// TIA Portal project "test" (V15.1)
// Vorlageprojekt für das Buch mit Zielsystem S7-1200

(* hardware
DEVICE "S7-1200-Station_1"  S7-1200 Station
   slot 0: "Baugruppenträger_0"  Rack  V1.0
   slot 1: "PLC_1"  CPU 1211C DC/DC/DC  6ES7 211-1AE40-0XB0  V4.1
*)

// ===== PLC "PLC_1"  CPU 1211C DC/DC/DC =====

VAR_GLOBAL   // PLC tag table "Standard-Variablentabelle"
   "Đèn báo hệ thống" AT %A0.0 : Bool;
   "START" AT %E0.0 : Bool;
   "STOP" AT %E0.1 : Bool;
   "Fill_1" AT %QD30 : Real;
   "Cb1" AT %I1.3 : Bool;
   "Lv_1_analog" AT %ID30 : DWord;
   "TG_Run1" AT %M0.0 : Bool;
   "ena_fill_1" AT %M3.0 : Bool;
   "Lv_2_analog" AT %ID34 : DWord;
   "TG_Cb1" AT %M1.3 : Bool;
   "ena_fill_2" AT %M3.4 : Bool;
   "Bt1" AT %Q1.3 : Bool;
   "Fill_2" AT %QD34 : Real;
   "TG_Fill_1" AT %MD30 : Real;
   "TG_Fill_2" AT %MD34 : Real;
   "TG_Fill_3" AT %MD40 : DWord;
   "V3_Calculate_1" AT %MD42 : DWord;
   "Set xa 1" AT %ID38 : Real;
   "Display xa 1" AT %QD54 : DInt;
   "Tag_14" AT %MD54 : DInt;
   "Set xa 2" AT %ID42 : Real;
   "Display xa 2" AT %QD58 : DInt;
   "Level_1" AT %MD10 : Real;
   "TG_Xa1+Xa2" AT %MD0 : DInt;
   "TG_Weight" AT %MD26 : DWord;
   "V3_Calculate" AT %MD38 : Real;
   "V1" AT %MD48 : Real;
   "V2" AT %MD52 : Real;
   "Start_tron" AT %I0.2 : Bool;
   "Tag_1" AT %MW0 : Int;
   "ĐK_Dis_1_2" AT %M1.2 : Bool;
   "Đèn_Trộn_Vàng" AT %Q0.1 : Bool;
   "Red light" AT %Q0.2 : Bool;
   "V3" AT %MD56 : Real;
   "Lv_3_analog" AT %ID46 : Real;
   "Fill_3" AT %QD38 : DWord;
   "TG_Tron_3" AT %M0.2 : Bool;
   "ena_fill_3" AT %M3.6 : Bool;
   "TG_Set1" AT %MD46 : Real;
   "Level_3" AT %MD6 : DInt;
   "Level_2" AT %MD8 : Real;
   "V1_Calculate" AT %MD12 : Real;
   "V2_Calculate" AT %MD16 : Real;
   "Discharge 1" AT %QD42 : Real;
   "Discharge 2" AT %QD46 : Real;
   "ena_discharge_1_2" AT %M3.7 : Bool;
   "TG_Xa_1_2" AT %M0.3 : Bool;
   "Cvey_Weight_1" AT %Q0.5 : Bool;
   "Weight 1" AT %ID50 : Real;
   "m3_Obj_1" AT %MD20 : Real;
   "Discharge 3" AT %QD50 : Real;
   "Start_Chiet" AT %M4.0 : Bool;
   "TG Dis 3" AT %MD50 : Real;
   "Continue with 10kg" AT %M4.1 : Bool;
   "V3_after" AT %MD44 : Real;
   "m3_before" AT %MD58 : DInt;
   "V3_bđầu" AT %MD4 : Real;
   "Tag_3" AT %M5.5 : Bool;
   "Tag_4" AT %M5.6 : Bool;
   "bt2" AT %Q1.4 : Bool;
   "bt3" AT %Q1.5 : Bool;
   "bt4" AT %Q1.6 : Bool;
   "bt5" AT %Q1.7 : Bool;
   "Tag_7" AT %MD28 : DWord;
   "Cb 2" AT %I1.4 : Bool;
   "Tag_9" AT %M10.2 : Bool;
   "Tag_10" AT %MB10 : Byte;
   "Tag_11" AT %M11.0 : Bool;
   "Tag_12" AT %M8.0 : Bool;
   "Tag_15" AT %M20.0 : Bool;
   "Tag_16" AT %M50.0 : Bool;
   "Tag_17" AT %M50.1 : Bool;
   "Wheel On" AT %Q0.6 : Bool;
   "Wheel Left" AT %Q0.7 : Bool;
   "Wheel Right" AT %Q1.0 : Bool;
   "Tag_21" AT %I6.0 : Bool;
   "Tag_22" AT %I6.1 : Bool;
   "Tag_23" AT %M8.5 : Bool;
   "Tag_25" AT %M50.2 : Bool;
   "Tag_26" AT %M50.3 : Bool;
   "Tag_27" AT %M70.1 : Bool;
   "Tag_28" AT %M70.2 : Bool;
   "Cvey_Weight_2" AT %Q0.4 : Bool;
   "Weight 2" AT %ID54 : Real;
   "m3_Obj_2" AT %MD22 : Real;
   "Tag_29" AT %M1.4 : Bool;
   "Tag_30" AT %MW50 : Int;
   "10kg" AT %M40.0 : Bool;
   "15Kg(1)" AT %M40.1 : Bool;
   "Tag_5" AT %M60.0 : Bool;
   "Tag_13" AT %M60.1 : Bool;
   "Tag_18" AT %M60.2 : Bool;
   "Continue with 15kg" AT %M4.2 : Bool;
   "Tag_20" AT %MW30 : Int;
   "STOP when low" AT %M4.3 : Bool;
END_VAR

DATA_BLOCK "ConV Height Volume_DB"   // DB1
{ S7_Optimized_Access := 'TRUE' }
VERSION : 0.1
// stored: InstanceOfName ConV Height Volume
"ConV Height Volume"
BEGIN
END_DATA_BLOCK

DATA_BLOCK "Speed V1 V2_DB"   // DB2
{ S7_Optimized_Access := 'TRUE' }
VERSION : 0.1
// stored: InstanceOfName Speed V1 V2
"Speed V1 V2"
BEGIN
END_DATA_BLOCK

DATA_BLOCK "Dieu kien_DB"   // DB4
{ S7_Optimized_Access := 'TRUE' }
VERSION : 0.1
// stored: InstanceOfName Dieu kien
"Dieu kien"
BEGIN
END_DATA_BLOCK

DATA_BLOCK "Speed V3_DB"   // DB5
{ S7_Optimized_Access := 'TRUE' }
VERSION : 0.1
// stored: InstanceOfName Speed V3
"Speed V3"
BEGIN
END_DATA_BLOCK

// folder: System blocks/Program resources

DATA_BLOCK "T2"   // DB7
{ S7_Optimized_Access := 'TRUE' }
AUTHOR : Simatic
FAMILY : IEC
NAME : IEC_TMR
VERSION : 1.0
// stored: InstanceOfName IEC_TIMER
"IEC_TIMER"
BEGIN
END_DATA_BLOCK

DATA_BLOCK "T3"   // DB8
{ S7_Optimized_Access := 'TRUE' }
AUTHOR : Simatic
FAMILY : IEC
NAME : IEC_TMR
VERSION : 1.0
// stored: InstanceOfName IEC_TIMER
"IEC_TIMER"
BEGIN
END_DATA_BLOCK

// folder: (top level)

FUNCTION_BLOCK "ConV Height Volume"   // FB1, LAD
{ S7_Optimized_Access := 'TRUE' }
VERSION : 0.1
   VAR_INPUT
      AnalogInput1 : Real;
      AnalogInput2 : Real;
      AnalogInput3 : Real;
   END_VAR
   VAR_OUTPUT
      RealLevel1 : Real;
      RealLevel2 : Real;
      RealLevel3 : Real;
      V1 : Real;
      V2 : Real;
      V3 : Real;
   END_VAR
   VAR_TEMP
      AnalogTemp1 : Real;
      AnalogTemp2 : Real;
      AnalogTemp3 : Real;
   END_VAR
BEGIN

REGION Network 1
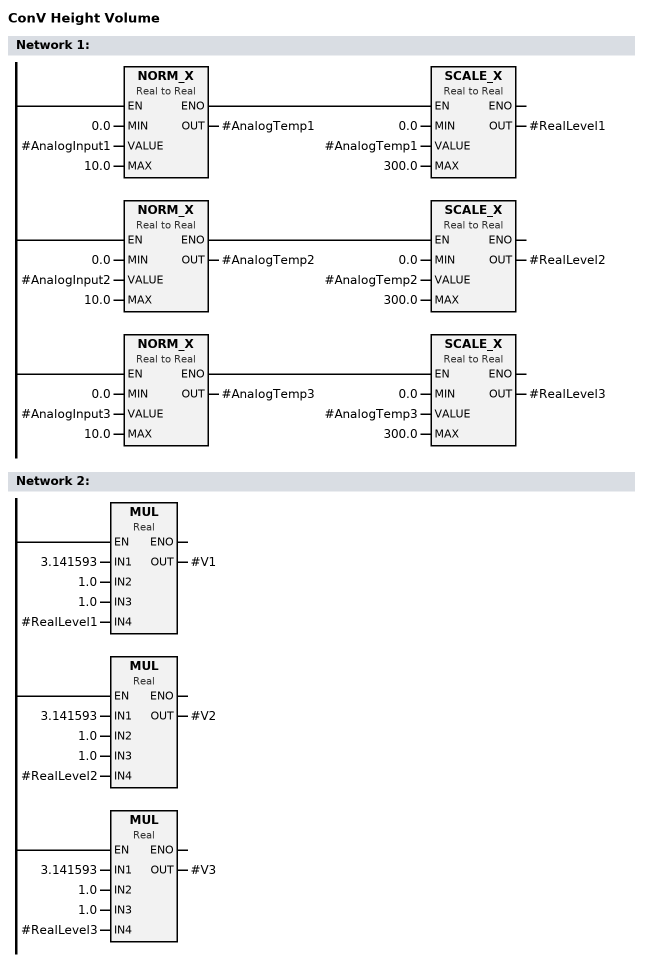
   RUNG wire#powerrail
      { S7_Templates := "[SrcType := Real, DestType := Real]" } Normalize(min := 0.0, value := #AnalogInput1, max := 10.0, out => #AnalogTemp1)
      { S7_Templates := "[SrcType := Real, DestType := Real]" } Scale(min := 0.0, value := #AnalogTemp1, max := 300.0, out => #RealLevel1)
   END_RUNG
   RUNG wire#powerrail
      { S7_Templates := "[SrcType := Real, DestType := Real]" } Normalize(min := 0.0, value := #AnalogInput2, max := 10.0, out => #AnalogTemp2)
      { S7_Templates := "[SrcType := Real, DestType := Real]" } Scale(min := 0.0, value := #AnalogTemp2, max := 300.0, out => #RealLevel2)
   END_RUNG
   RUNG wire#powerrail
      { S7_Templates := "[SrcType := Real, DestType := Real]" } Normalize(min := 0.0, value := #AnalogInput3, max := 10.0, out => #AnalogTemp3)
      { S7_Templates := "[SrcType := Real, DestType := Real]" } Scale(min := 0.0, value := #AnalogTemp3, max := 300.0, out => #RealLevel3)
   END_RUNG
   // the same network as SCL:
   #AnalogTemp1 := NORM_X(MIN := 0.0, VALUE := #AnalogInput1, MAX := 10.0);
   #RealLevel1 := SCALE_X(MIN := 0.0, VALUE := #AnalogTemp1, MAX := 300.0);
   #AnalogTemp2 := NORM_X(MIN := 0.0, VALUE := #AnalogInput2, MAX := 10.0);
   #RealLevel2 := SCALE_X(MIN := 0.0, VALUE := #AnalogTemp2, MAX := 300.0);
   #AnalogTemp3 := NORM_X(MIN := 0.0, VALUE := #AnalogInput3, MAX := 10.0);
   #RealLevel3 := SCALE_X(MIN := 0.0, VALUE := #AnalogTemp3, MAX := 300.0);
END_REGION

REGION Network 2
   RUNG wire#powerrail
      { S7_Templates := "SrcType := Real" } Mul(in1 := 3.141593, in2 := 1.0, in3 := 1.0, in4 := #RealLevel1, out => #V1)
   END_RUNG
   RUNG wire#powerrail
      { S7_Templates := "SrcType := Real" } Mul(in1 := 3.141593, in2 := 1.0, in3 := 1.0, in4 := #RealLevel2, out => #V2)
   END_RUNG
   RUNG wire#powerrail
      { S7_Templates := "SrcType := Real" } Mul(in1 := 3.141593, in2 := 1.0, in3 := 1.0, in4 := #RealLevel3, out => #V3)
   END_RUNG
   // the same network as SCL:
   #V1 := 3.141593 * 1.0 * 1.0 * #RealLevel1;
   #V2 := 3.141593 * 1.0 * 1.0 * #RealLevel2;
   #V3 := 3.141593 * 1.0 * 1.0 * #RealLevel3;
END_REGION
END_FUNCTION_BLOCK

FUNCTION_BLOCK "Dieu kien"   // FB2, LAD
{ S7_Optimized_Access := 'TRUE' }
VERSION : 0.1
   VAR_INPUT
      Display_xa_1 : DInt;
      Display_xa_2 : DInt;
   END_VAR
   VAR_OUTPUT
      V3_calculate : Real;
      V1_Cal : Real;
      V2_Cal : Real;
   END_VAR
   VAR_TEMP
      "int1+int2" : DInt;
      dk1 : Real;   // 100
      dk2 : Real;   // 942.4777 - Thể tích max
      V3_calculate_1 : Real;
      V1_calculate : Real;
      V2_calculate : Real;
   END_VAR
   VAR_TEMP   // added for the SCL form of the ladder/FBD networks
      _w1 : Bool;
      _w2 : Bool;
   END_VAR
BEGIN

REGION Network 1
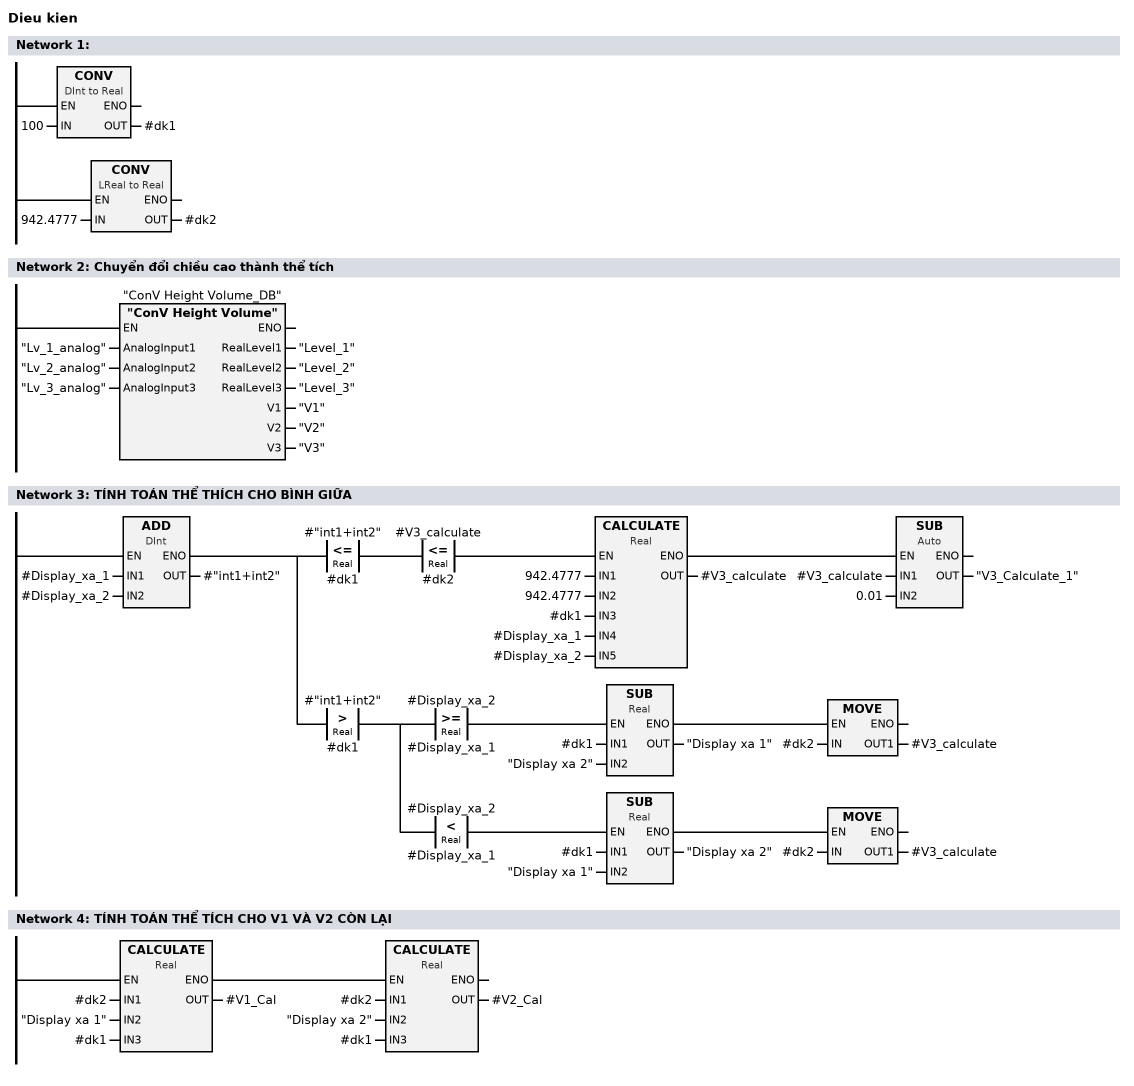
   RUNG wire#powerrail
      { S7_Templates := "[SrcType := DInt, DestType := Real]" } Convert(in := 100, out => #dk1)
   END_RUNG
   RUNG wire#powerrail
      { S7_Templates := "[SrcType := LReal, DestType := Real]" } Convert(in := 942.4777, out => #dk2)
   END_RUNG
   // the same network as SCL:
   #dk1 := DINT_TO_REAL(100);
   #dk2 := LREAL_TO_REAL(942.4777);
END_REGION

REGION Network 2: Chuyển đổi chiều cao thành thể tích
   RUNG wire#powerrail
      "ConV Height Volume_DB"(AnalogInput1 := "Lv_1_analog", AnalogInput2 := "Lv_2_analog", AnalogInput3 := "Lv_3_analog", RealLevel1 => "Level_1", RealLevel2 => "Level_2", RealLevel3 => "Level_3", V1 => "V1", V2 => "V2", V3 => "V3")
   END_RUNG
   // the same network as SCL:
   "ConV Height Volume_DB"(AnalogInput1 := "Lv_1_analog",   // "ConV Height Volume"
                           AnalogInput2 := "Lv_2_analog",
                           AnalogInput3 := "Lv_3_analog",
                           RealLevel1 => "Level_1",
                           RealLevel2 => "Level_2",
                           RealLevel3 => "Level_3",
                           V1 => "V1",
                           V2 => "V2",
                           V3 => "V3");
END_REGION

REGION Network 3: TÍNH TOÁN THỂ THÍCH CHO BÌNH GIỮA
   RUNG wire#powerrail
      { S7_Templates := "SrcType := DInt" } Add(in1 := #Display_xa_1, in2 := #Display_xa_2, out => #"int1+int2")
      wire#w1
      { S7_Templates := "SrcType := Real" } LE_Contact(in1 := #"int1+int2", in2 := #dk1)
      { S7_Templates := "SrcType := Real" } LE_Contact(in1 := #V3_calculate, in2 := #dk2)
      { S7_Templates := "SrcType := Real"; S7_Expression := "IN1*IN4/IN3+IN2*IN5/IN3" } Calculate(in1 := 942.4777, in2 := 942.4777, in3 := #dk1, in4 := #Display_xa_1, in5 := #Display_xa_2, out => #V3_calculate)
      Sub(in1 := #V3_calculate, in2 := 0.01, out => "V3_Calculate_1")
   END_RUNG
   RUNG wire#w1
      { S7_Templates := "SrcType := Real" } GT_Contact(in1 := #"int1+int2", in2 := #dk1)
      wire#w2
      { S7_Templates := "SrcType := Real" } GE_Contact(in1 := #Display_xa_2, in2 := #Display_xa_1)
      { S7_Templates := "SrcType := Real" } Sub(in1 := #dk1, in2 := "Display xa 2", out => "Display xa 1")
      Move(in := #dk2, out1 => #V3_calculate)
   END_RUNG
   RUNG wire#w2
      { S7_Templates := "SrcType := Real" } LT_Contact(in1 := #Display_xa_2, in2 := #Display_xa_1)
      { S7_Templates := "SrcType := Real" } Sub(in1 := #dk1, in2 := "Display xa 1", out => "Display xa 2")
      Move(in := #dk2, out1 => #V3_calculate)
   END_RUNG
   // the same network as SCL:
   #"int1+int2" := #Display_xa_1 + #Display_xa_2;
   #_w1 := (#"int1+int2" <= #dk1) AND (#V3_calculate <= #dk2);
   IF #_w1 THEN
       #V3_calculate := 942.4777*#Display_xa_1/#dk1+942.4777*#Display_xa_2/#dk1;
       "V3_Calculate_1" := #V3_calculate - 0.01;
   END_IF;
   #_w2 := #"int1+int2" > #dk1;
   IF #_w2 AND (#Display_xa_2 >= #Display_xa_1) THEN
       "Display xa 1" := #dk1 - "Display xa 2";
       #V3_calculate := #dk2;
   END_IF;
   IF #_w2 AND (#Display_xa_2 < #Display_xa_1) THEN
       "Display xa 2" := #dk1 - "Display xa 1";
       #V3_calculate := #dk2;
   END_IF;
END_REGION

REGION Network 4: TÍNH TOÁN THỂ TÍCH CHO V1 VÀ V2 CÒN LẠI
   RUNG wire#powerrail
      { S7_Templates := "SrcType := Real"; S7_Expression := "(IN1-IN2*IN1/IN3)" } Calculate(in1 := #dk2, in2 := "Display xa 1", in3 := #dk1, out => #V1_Cal)
      { S7_Templates := "SrcType := Real"; S7_Expression := "(IN1-IN2*IN1/IN3)" } Calculate(in1 := #dk2, in2 := "Display xa 2", in3 := #dk1, out => #V2_Cal)
   END_RUNG
   // the same network as SCL:
   #V1_Cal := (#dk2-"Display xa 1"*#dk2/#dk1);
   #V2_Cal := (#dk2-"Display xa 2"*#dk2/#dk1);
END_REGION
END_FUNCTION_BLOCK

FUNCTION_BLOCK "Speed V3"   // FB3, LAD
{ S7_Optimized_Access := 'TRUE' }
VERSION : 0.1
   VAR_OUTPUT
      "Speed Fill 3" : Real;
   END_VAR
   VAR_TEMP
      dk1 : DInt;   // 150
      hs1 : DInt;   // 490
      dk2 : DInt;   // 295
      hs2 : DInt;   // 10
      Temp_1 : DInt;
      "Speed Fill 3 Dint" : Real;
      V3_Calculate : Real;
   END_VAR
BEGIN

REGION Network 1
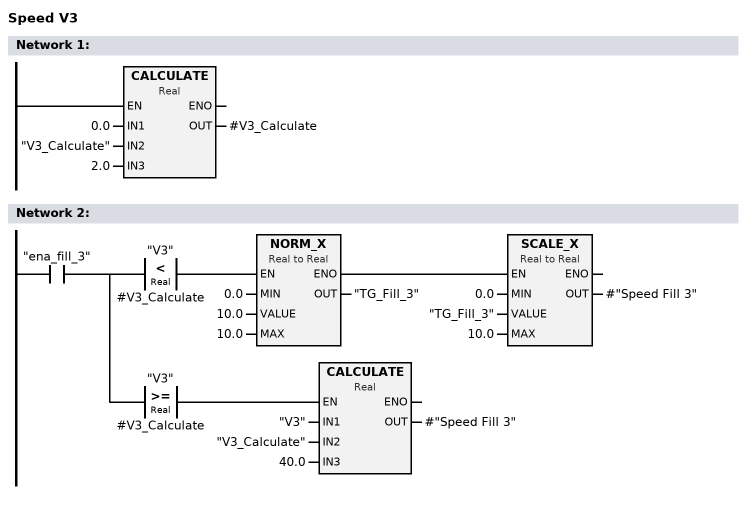
   RUNG wire#powerrail
      { S7_Templates := "SrcType := Real"; S7_Expression := "(IN2-IN1)/IN3" } Calculate(in1 := 0.0, in2 := "V3_Calculate", in3 := 2.0, out => #V3_Calculate)
   END_RUNG
   // the same network as SCL:
   #V3_Calculate := ("V3_Calculate"-0.0)/2.0;
END_REGION

REGION Network 2
   RUNG wire#powerrail
      Contact( "ena_fill_3" )
      wire#w1
      { S7_Templates := "SrcType := Real" } LT_Contact(in1 := "V3", in2 := #V3_Calculate)
      { S7_Templates := "[SrcType := Real, DestType := Real]" } Normalize(min := 0.0, value := 10.0, max := 10.0, out => "TG_Fill_3")
      { S7_Templates := "[SrcType := Real, DestType := Real]" } Scale(min := 0.0, value := "TG_Fill_3", max := 10.0, out => #"Speed Fill 3")
   END_RUNG
   RUNG wire#w1
      { S7_Templates := "SrcType := Real" } GE_Contact(in1 := "V3", in2 := #V3_Calculate)
      { S7_Templates := "SrcType := Real"; S7_Expression := "-IN3*IN1*IN1/(IN2*IN2)+IN3*IN1/IN2" } Calculate(in1 := "V3", in2 := "V3_Calculate", in3 := 40.0, out => #"Speed Fill 3")
   END_RUNG
   // the same network as SCL:
   IF "ena_fill_3" AND ("V3" < #V3_Calculate) THEN
       "TG_Fill_3" := NORM_X(MIN := 0.0, VALUE := 10.0, MAX := 10.0);
       #"Speed Fill 3" := SCALE_X(MIN := 0.0, VALUE := "TG_Fill_3", MAX := 10.0);
   END_IF;
   IF "ena_fill_3" AND ("V3" >= #V3_Calculate) THEN
       #"Speed Fill 3" := -40.0*"V3"*"V3"/("V3_Calculate"*"V3_Calculate")+40.0*"V3"/"V3_Calculate";
   END_IF;
END_REGION
END_FUNCTION_BLOCK

FUNCTION_BLOCK "Speed V1 V2"   // FB4, LAD
{ S7_Optimized_Access := 'TRUE' }
VERSION : 0.1
   VAR_OUTPUT
      "Speed dis 1" : Real;
      "Speed dis 2" : Real;
   END_VAR
   VAR_TEMP
      V1_Calculate : Real;
      V2_Calculate : Real;
      TG_Dis_1 : DWord;
      TG_Dis_2 : DWord;
   END_VAR
BEGIN

REGION Network 1
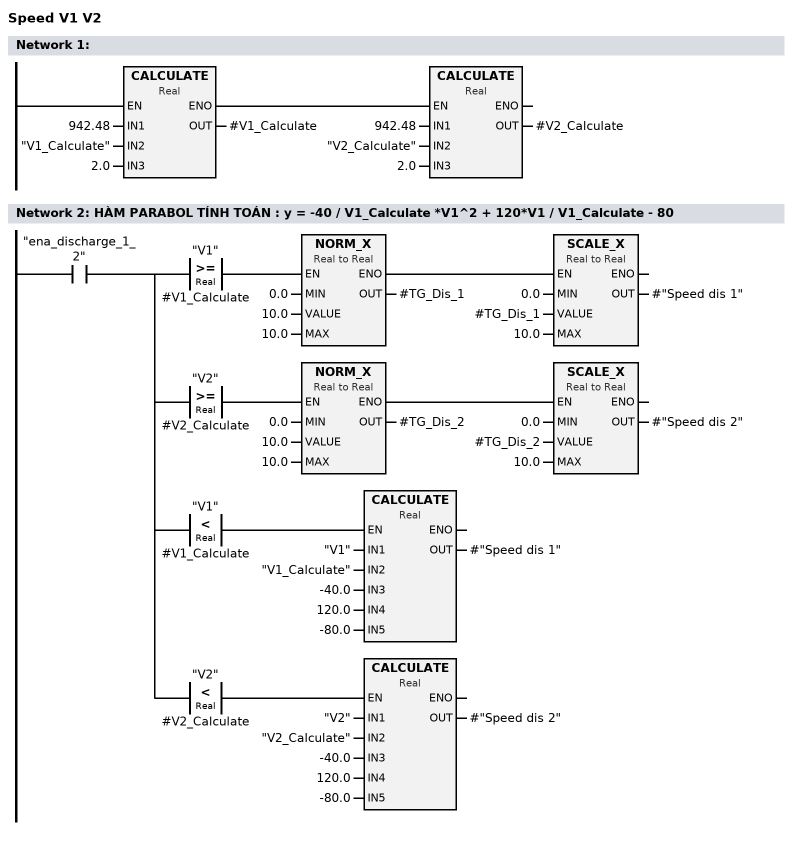
   RUNG wire#powerrail
      { S7_Templates := "SrcType := Real"; S7_Expression := "(IN1-IN2)/IN3+IN2" } Calculate(in1 := 942.48, in2 := "V1_Calculate", in3 := 2.0, out => #V1_Calculate)
      { S7_Templates := "SrcType := Real"; S7_Expression := "(IN1-IN2)/IN3+IN2" } Calculate(in1 := 942.48, in2 := "V2_Calculate", in3 := 2.0, out => #V2_Calculate)
   END_RUNG
   // the same network as SCL:
   #V1_Calculate := (942.48-"V1_Calculate")/2.0+"V1_Calculate";
   #V2_Calculate := (942.48-"V2_Calculate")/2.0+"V2_Calculate";
END_REGION

REGION Network 2: HÀM PARABOL TÍNH TOÁN : y = -40 / V1_Calculate *V1^2 + 120*V1 / V1_Calculate - 80
   RUNG wire#powerrail
      Contact( "ena_discharge_1_2" )
      wire#w1
      { S7_Templates := "SrcType := Real" } GE_Contact(in1 := "V1", in2 := #V1_Calculate)
      { S7_Templates := "[SrcType := Real, DestType := Real]" } Normalize(min := 0.0, value := 10.0, max := 10.0, out => #TG_Dis_1)
      { S7_Templates := "[SrcType := Real, DestType := Real]" } Scale(min := 0.0, value := #TG_Dis_1, max := 10.0, out => #"Speed dis 1")
   END_RUNG
   RUNG wire#w1
      { S7_Templates := "SrcType := Real" } GE_Contact(in1 := "V2", in2 := #V2_Calculate)
      { S7_Templates := "[SrcType := Real, DestType := Real]" } Normalize(min := 0.0, value := 10.0, max := 10.0, out => #TG_Dis_2)
      { S7_Templates := "[SrcType := Real, DestType := Real]" } Scale(min := 0.0, value := #TG_Dis_2, max := 10.0, out => #"Speed dis 2")
   END_RUNG
   RUNG wire#w1
      { S7_Templates := "SrcType := Real" } LT_Contact(in1 := "V1", in2 := #V1_Calculate)
      { S7_Templates := "SrcType := Real"; S7_Expression := "IN3/(IN2*IN2)*IN1*IN1+IN4*IN1/IN2+IN5" } Calculate(in1 := "V1", in2 := "V1_Calculate", in3 := -40.0, in4 := 120.0, in5 := -80.0, out => #"Speed dis 1")
   END_RUNG
   RUNG wire#w1
      { S7_Templates := "SrcType := Real" } LT_Contact(in1 := "V2", in2 := #V2_Calculate)
      { S7_Templates := "SrcType := Real"; S7_Expression := "IN3/(IN2*IN2)*IN1*IN1+IN4*IN1/IN2+IN5" } Calculate(in1 := "V2", in2 := "V2_Calculate", in3 := -40.0, in4 := 120.0, in5 := -80.0, out => #"Speed dis 2")
   END_RUNG
   // the same network as SCL:
   IF "ena_discharge_1_2" AND ("V1" >= #V1_Calculate) THEN
       #TG_Dis_1 := NORM_X(MIN := 0.0, VALUE := 10.0, MAX := 10.0);
       #"Speed dis 1" := SCALE_X(MIN := 0.0, VALUE := #TG_Dis_1, MAX := 10.0);
   END_IF;
   IF "ena_discharge_1_2" AND ("V2" >= #V2_Calculate) THEN
       #TG_Dis_2 := NORM_X(MIN := 0.0, VALUE := 10.0, MAX := 10.0);
       #"Speed dis 2" := SCALE_X(MIN := 0.0, VALUE := #TG_Dis_2, MAX := 10.0);
   END_IF;
   IF "ena_discharge_1_2" AND ("V1" < #V1_Calculate) THEN
       #"Speed dis 1" := (-40.0)/("V1_Calculate"*"V1_Calculate")*"V1"*"V1"+120.0*"V1"/"V1_Calculate"+(-80.0);
   END_IF;
   IF "ena_discharge_1_2" AND ("V2" < #V2_Calculate) THEN
       #"Speed dis 2" := (-40.0)/("V2_Calculate"*"V2_Calculate")*"V2"*"V2"+120.0*"V2"/"V2_Calculate"+(-80.0);
   END_IF;
END_REGION
END_FUNCTION_BLOCK

FUNCTION "Run" : Void   // FC1, LAD
{ S7_Optimized_Access := 'TRUE' }
VERSION : 0.1
BEGIN

REGION Network 1
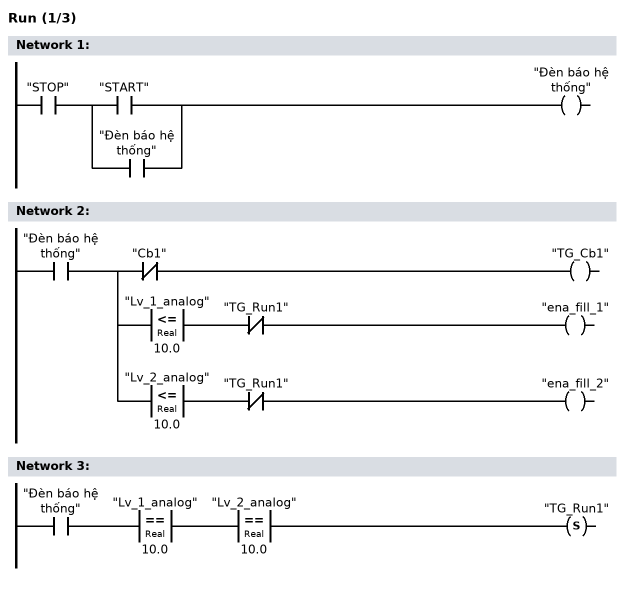
   RUNG wire#powerrail
      Contact( "STOP" )
      wire#w1
      Contact( "START" )
      wire#w2
      Coil( "Đèn báo hệ thống" )
   END_RUNG
   RUNG wire#w1
      Contact( "Đèn báo hệ thống" )
   END_RUNG wire#w2
   // the same network as SCL:
   "Đèn báo hệ thống" := "STOP" AND ("START" OR "Đèn báo hệ thống");
END_REGION

REGION Network 2
   RUNG wire#powerrail
      Contact( "Đèn báo hệ thống" )
      wire#w1
      I_Contact( "Cb1" )
      Coil( "TG_Cb1" )
   END_RUNG
   RUNG wire#w1
      { S7_Templates := "SrcType := Real" } LE_Contact(in1 := "Lv_1_analog", in2 := 10.0)
      I_Contact( "TG_Run1" )
      Coil( "ena_fill_1" )
   END_RUNG
   RUNG wire#w1
      { S7_Templates := "SrcType := Real" } LE_Contact(in1 := "Lv_2_analog", in2 := 10.0)
      I_Contact( "TG_Run1" )
      Coil( "ena_fill_2" )
   END_RUNG
   // the same network as SCL:
   "TG_Cb1" := "Đèn báo hệ thống" AND NOT "Cb1";
   "ena_fill_1" := "Đèn báo hệ thống" AND ("Lv_1_analog" <= 10.0) AND NOT "TG_Run1";
   "ena_fill_2" := "Đèn báo hệ thống" AND ("Lv_2_analog" <= 10.0) AND NOT "TG_Run1";
END_REGION

REGION Network 3
   RUNG wire#powerrail
      Contact( "Đèn báo hệ thống" )
      { S7_Templates := "SrcType := Real" } EQ_Contact(in1 := "Lv_1_analog", in2 := 10.0)
      { S7_Templates := "SrcType := Real" } EQ_Contact(in1 := "Lv_2_analog", in2 := 10.0)
      S_Coil( "TG_Run1" )
   END_RUNG
   // the same network as SCL:
   IF "Đèn báo hệ thống" AND ("Lv_1_analog" = 10.0) AND ("Lv_2_analog" = 10.0) THEN
       "TG_Run1" := TRUE;
   END_IF;
END_REGION

REGION Network 4
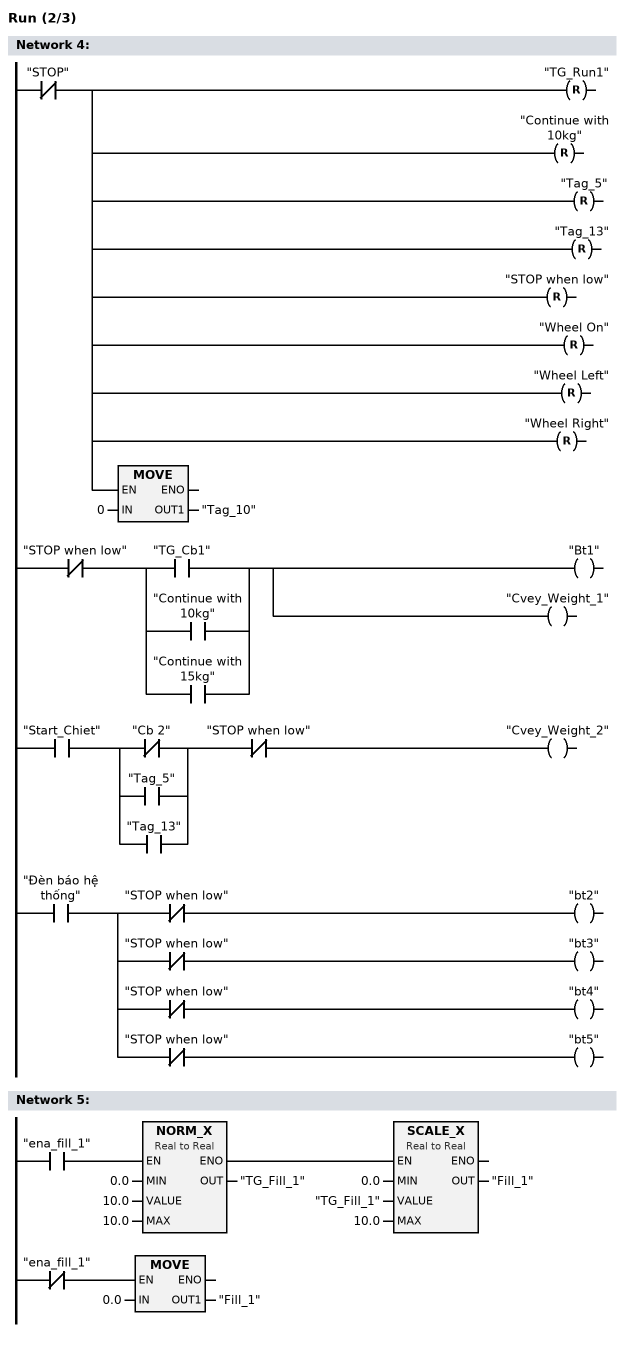
   RUNG wire#powerrail
      I_Contact( "STOP" )
      wire#w1
      R_Coil( "TG_Run1" )
   END_RUNG
   RUNG wire#w1
      R_Coil( "Continue with 10kg" )
   END_RUNG
   RUNG wire#w1
      R_Coil( "Tag_5" )
   END_RUNG
   RUNG wire#w1
      R_Coil( "Tag_13" )
   END_RUNG
   RUNG wire#w1
      R_Coil( "STOP when low" )
   END_RUNG
   RUNG wire#w1
      R_Coil( "Wheel On" )
   END_RUNG
   RUNG wire#w1
      R_Coil( "Wheel Left" )
   END_RUNG
   RUNG wire#w1
      R_Coil( "Wheel Right" )
   END_RUNG
   RUNG wire#w1
      Move(in := 0, out1 => "Tag_10")
   END_RUNG
   RUNG wire#powerrail
      I_Contact( "STOP when low" )
      wire#w2
      Contact( "TG_Cb1" )
      wire#w3
      Coil( "Bt1" )
   END_RUNG
   RUNG wire#w2
      Contact( "Continue with 10kg" )
   END_RUNG wire#w3
   RUNG wire#w2
      Contact( "Continue with 15kg" )
   END_RUNG wire#w3
   RUNG wire#w3
      Coil( "Cvey_Weight_1" )
   END_RUNG
   RUNG wire#powerrail
      Contact( "Start_Chiet" )
      wire#w4
      I_Contact( "Cb 2" )
      wire#w5
      I_Contact( "STOP when low" )
      Coil( "Cvey_Weight_2" )
   END_RUNG
   RUNG wire#w4
      Contact( "Tag_5" )
   END_RUNG wire#w5
   RUNG wire#w4
      Contact( "Tag_13" )
   END_RUNG wire#w5
   RUNG wire#powerrail
      Contact( "Đèn báo hệ thống" )
      wire#w6
      I_Contact( "STOP when low" )
      Coil( "bt2" )
   END_RUNG
   RUNG wire#w6
      I_Contact( "STOP when low" )
      Coil( "bt3" )
   END_RUNG
   RUNG wire#w6
      I_Contact( "STOP when low" )
      Coil( "bt4" )
   END_RUNG
   RUNG wire#w6
      I_Contact( "STOP when low" )
      Coil( "bt5" )
   END_RUNG
   // the same network as SCL:
   IF NOT "STOP" THEN
       "TG_Run1" := FALSE;
       "Continue with 10kg" := FALSE;
       "Tag_5" := FALSE;
       "Tag_13" := FALSE;
       "STOP when low" := FALSE;
       "Wheel On" := FALSE;
       "Wheel Left" := FALSE;
       "Wheel Right" := FALSE;
       "Tag_10" := 0;
   END_IF;
   "Bt1" := NOT "STOP when low" AND ("TG_Cb1" OR "Continue with 10kg" OR "Continue with 15kg");
   "Cvey_Weight_1" := "Bt1";
   "Cvey_Weight_2" := "Start_Chiet" AND (NOT "Cb 2" OR "Tag_5" OR "Tag_13") AND NOT "STOP when low";
   "bt2" := "Đèn báo hệ thống" AND NOT "STOP when low";
   "bt3" := "Đèn báo hệ thống" AND NOT "STOP when low";
   "bt4" := "Đèn báo hệ thống" AND NOT "STOP when low";
   "bt5" := "Đèn báo hệ thống" AND NOT "STOP when low";
END_REGION

REGION Network 5
   RUNG wire#powerrail
      Contact( "ena_fill_1" )
      { S7_Templates := "[SrcType := Real, DestType := Real]" } Normalize(min := 0.0, value := 10.0, max := 10.0, out => "TG_Fill_1")
      { S7_Templates := "[SrcType := Real, DestType := Real]" } Scale(min := 0.0, value := "TG_Fill_1", max := 10.0, out => "Fill_1")
   END_RUNG
   RUNG wire#powerrail
      I_Contact( "ena_fill_1" )
      Move(in := 0.0, out1 => "Fill_1")
   END_RUNG
   // the same network as SCL:
   IF "ena_fill_1" THEN
       "TG_Fill_1" := NORM_X(MIN := 0.0, VALUE := 10.0, MAX := 10.0);
       "Fill_1" := SCALE_X(MIN := 0.0, VALUE := "TG_Fill_1", MAX := 10.0);
   END_IF;
   IF NOT "ena_fill_1" THEN "Fill_1" := 0.0; END_IF;
END_REGION

REGION Network 6
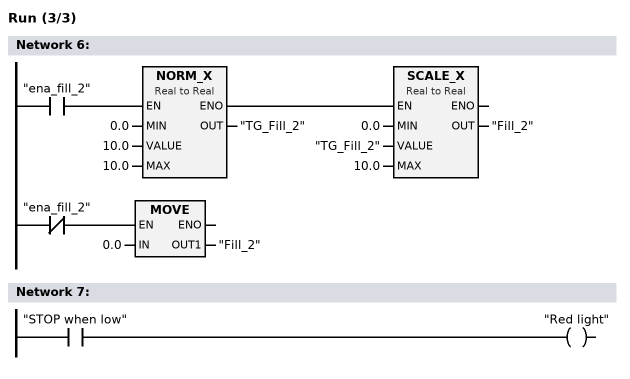
   RUNG wire#powerrail
      Contact( "ena_fill_2" )
      { S7_Templates := "[SrcType := Real, DestType := Real]" } Normalize(min := 0.0, value := 10.0, max := 10.0, out => "TG_Fill_2")
      { S7_Templates := "[SrcType := Real, DestType := Real]" } Scale(min := 0.0, value := "TG_Fill_2", max := 10.0, out => "Fill_2")
   END_RUNG
   RUNG wire#powerrail
      I_Contact( "ena_fill_2" )
      Move(in := 0.0, out1 => "Fill_2")
   END_RUNG
   // the same network as SCL:
   IF "ena_fill_2" THEN
       "TG_Fill_2" := NORM_X(MIN := 0.0, VALUE := 10.0, MAX := 10.0);
       "Fill_2" := SCALE_X(MIN := 0.0, VALUE := "TG_Fill_2", MAX := 10.0);
   END_IF;
   IF NOT "ena_fill_2" THEN "Fill_2" := 0.0; END_IF;
END_REGION

REGION Network 7
   RUNG wire#powerrail
      Contact( "STOP when low" )
      Coil( "Red light" )
   END_RUNG
   // the same network as SCL:
   "Red light" := "STOP when low";
END_REGION
END_FUNCTION

FUNCTION "Tron" : Void   // FC2, LAD
{ S7_Optimized_Access := 'TRUE' }
VERSION : 0.1
   VAR_TEMP   // added for the SCL form of the ladder/FBD networks
      _w1 : Bool;
   END_VAR
BEGIN

REGION Network 1
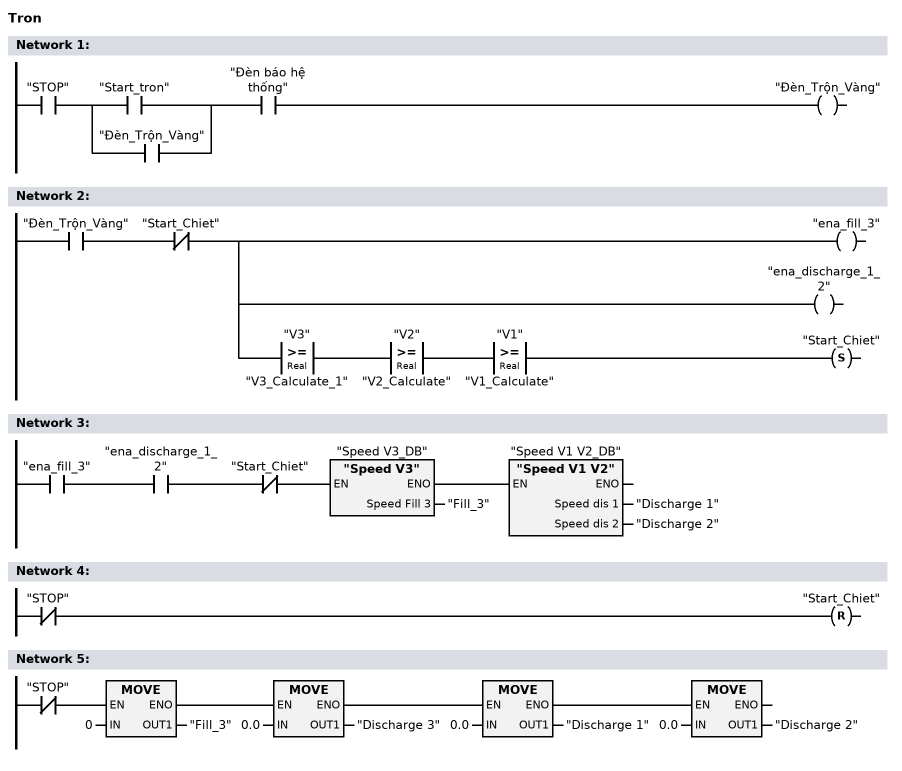
   RUNG wire#powerrail
      Contact( "STOP" )
      wire#w1
      Contact( "Start_tron" )
      wire#w2
      Contact( "Đèn báo hệ thống" )
      Coil( "Đèn_Trộn_Vàng" )
   END_RUNG
   RUNG wire#w1
      Contact( "Đèn_Trộn_Vàng" )
   END_RUNG wire#w2
   // the same network as SCL:
   "Đèn_Trộn_Vàng" := "STOP" AND ("Start_tron" OR "Đèn_Trộn_Vàng") AND "Đèn báo hệ thống";
END_REGION

REGION Network 2
   RUNG wire#powerrail
      Contact( "Đèn_Trộn_Vàng" )
      I_Contact( "Start_Chiet" )
      wire#w1
      Coil( "ena_fill_3" )
   END_RUNG
   RUNG wire#w1
      Coil( "ena_discharge_1_2" )
   END_RUNG
   RUNG wire#w1
      { S7_Templates := "SrcType := Real" } GE_Contact(in1 := "V3", in2 := "V3_Calculate_1")
      { S7_Templates := "SrcType := Real" } GE_Contact(in1 := "V2", in2 := "V2_Calculate")
      { S7_Templates := "SrcType := Real" } GE_Contact(in1 := "V1", in2 := "V1_Calculate")
      S_Coil( "Start_Chiet" )
   END_RUNG
   // the same network as SCL:
   "ena_fill_3" := "Đèn_Trộn_Vàng" AND NOT "Start_Chiet";
   "ena_discharge_1_2" := "ena_fill_3";
   IF "ena_fill_3" AND ("V3" >= "V3_Calculate_1") AND ("V2" >= "V2_Calculate") AND ("V1" >= "V1_Calculate") THEN
       "Start_Chiet" := TRUE;
   END_IF;
END_REGION

REGION Network 3
   RUNG wire#powerrail
      Contact( "ena_fill_3" )
      Contact( "ena_discharge_1_2" )
      I_Contact( "Start_Chiet" )
      "Speed V3_DB"("Speed Fill 3" => "Fill_3")
      "Speed V1 V2_DB"("Speed dis 1" => "Discharge 1", "Speed dis 2" => "Discharge 2")
   END_RUNG
   // the same network as SCL:
   "Speed V3_DB"(EN := "ena_fill_3" AND "ena_discharge_1_2" AND NOT "Start_Chiet",   // "Speed V3"
                 "Speed Fill 3" => "Fill_3",
                 ENO => #_w1);
   IF #_w1 THEN
       "Speed V1 V2_DB"("Speed dis 1" => "Discharge 1", "Speed dis 2" => "Discharge 2");   // "Speed V1 V2"
   END_IF;
END_REGION

REGION Network 4
   RUNG wire#powerrail
      I_Contact( "STOP" )
      R_Coil( "Start_Chiet" )
   END_RUNG
   // the same network as SCL:
   IF NOT "STOP" THEN "Start_Chiet" := FALSE; END_IF;
END_REGION

REGION Network 5
   RUNG wire#powerrail
      I_Contact( "STOP" )
      Move(in := 0, out1 => "Fill_3")
      Move(in := 0.0, out1 => "Discharge 3")
      Move(in := 0.0, out1 => "Discharge 1")
      Move(in := 0.0, out1 => "Discharge 2")
   END_RUNG
   // the same network as SCL:
   IF NOT "STOP" THEN
       "Fill_3" := 0;
       "Discharge 3" := 0.0;
       "Discharge 1" := 0.0;
       "Discharge 2" := 0.0;
   END_IF;
END_REGION
END_FUNCTION

FUNCTION "Hien thi muc Xa" : Void   // FC3, LAD
{ S7_Optimized_Access := 'TRUE' }
VERSION : 0.1
BEGIN

REGION Network 1
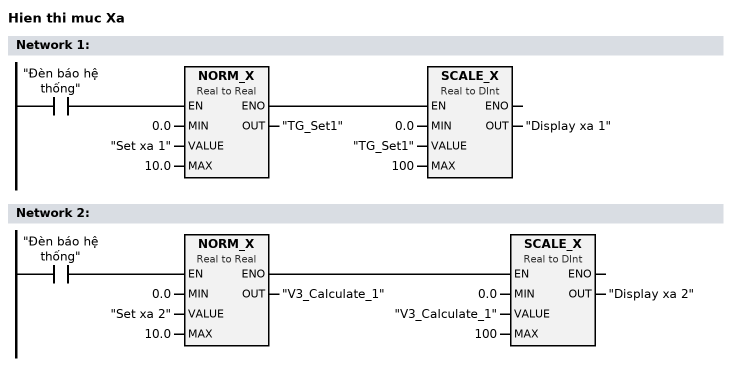
   RUNG wire#powerrail
      Contact( "Đèn báo hệ thống" )
      { S7_Templates := "[SrcType := Real, DestType := Real]" } Normalize(min := 0.0, value := "Set xa 1", max := 10.0, out => "TG_Set1")
      { S7_Templates := "[SrcType := Real, DestType := DInt]" } Scale(min := 0.0, value := "TG_Set1", max := 100, out => "Display xa 1")
   END_RUNG
   // the same network as SCL:
   IF "Đèn báo hệ thống" THEN
       "TG_Set1" := NORM_X(MIN := 0.0, VALUE := "Set xa 1", MAX := 10.0);
       "Display xa 1" := SCALE_X(MIN := 0.0, VALUE := "TG_Set1", MAX := 100);
   END_IF;
END_REGION

REGION Network 2
   RUNG wire#powerrail
      Contact( "Đèn báo hệ thống" )
      { S7_Templates := "[SrcType := Real, DestType := Real]" } Normalize(min := 0.0, value := "Set xa 2", max := 10.0, out => "V3_Calculate_1")
      { S7_Templates := "[SrcType := Real, DestType := DInt]" } Scale(min := 0.0, value := "V3_Calculate_1", max := 100, out => "Display xa 2")
   END_RUNG
   // the same network as SCL:
   IF "Đèn báo hệ thống" THEN
       "V3_Calculate_1" := NORM_X(MIN := 0.0, VALUE := "Set xa 2", MAX := 10.0);
       "Display xa 2" := SCALE_X(MIN := 0.0, VALUE := "V3_Calculate_1", MAX := 100);
   END_IF;
END_REGION
END_FUNCTION

FUNCTION "Sorting and fill" : Void   // FC4, LAD
{ S7_Optimized_Access := 'TRUE' }
VERSION : 0.1
   VAR_TEMP
      Obj_Weight_1 : Real;
      v3_After : Real;
      TG_Dis_3 : Real;
      Obj_Weight_2 : Real;
   END_VAR
   VAR_TEMP   // added for the SCL form of the ladder/FBD networks
      _w1 : Bool;
      _w2 : Bool;
      _w3 : Bool;
   END_VAR
BEGIN

REGION Network 1
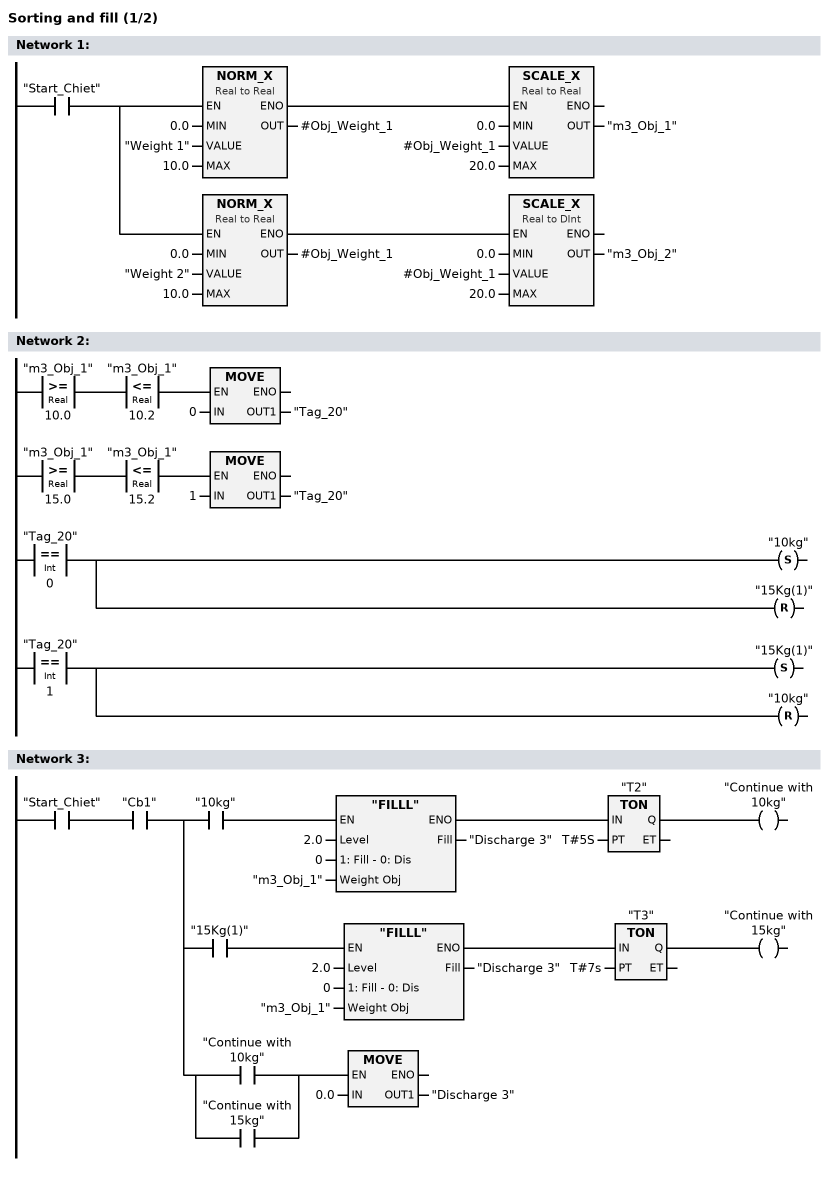
   RUNG wire#powerrail
      Contact( "Start_Chiet" )
      wire#w1
      { S7_Templates := "[SrcType := Real, DestType := Real]" } Normalize(min := 0.0, value := "Weight 1", max := 10.0, out => #Obj_Weight_1)
      { S7_Templates := "[SrcType := Real, DestType := Real]" } Scale(min := 0.0, value := #Obj_Weight_1, max := 20.0, out => "m3_Obj_1")
   END_RUNG
   RUNG wire#w1
      { S7_Templates := "[SrcType := Real, DestType := Real]" } Normalize(min := 0.0, value := "Weight 2", max := 10.0, out => #Obj_Weight_1)
      { S7_Templates := "[SrcType := Real, DestType := DInt]" } Scale(min := 0.0, value := #Obj_Weight_1, max := 20.0, out => "m3_Obj_2")
   END_RUNG
   // the same network as SCL:
   IF "Start_Chiet" THEN
       #Obj_Weight_1 := NORM_X(MIN := 0.0, VALUE := "Weight 1", MAX := 10.0);
       "m3_Obj_1" := SCALE_X(MIN := 0.0, VALUE := #Obj_Weight_1, MAX := 20.0);
       #Obj_Weight_1 := NORM_X(MIN := 0.0, VALUE := "Weight 2", MAX := 10.0);
       "m3_Obj_2" := SCALE_X(MIN := 0.0, VALUE := #Obj_Weight_1, MAX := 20.0);
   END_IF;
END_REGION

REGION Network 2
   RUNG wire#powerrail
      { S7_Templates := "SrcType := Real" } GE_Contact(in1 := "m3_Obj_1", in2 := 10.0)
      { S7_Templates := "SrcType := Real" } LE_Contact(in1 := "m3_Obj_1", in2 := 10.2)
      Move(in := 0, out1 => "Tag_20")
   END_RUNG
   RUNG wire#powerrail
      { S7_Templates := "SrcType := Real" } GE_Contact(in1 := "m3_Obj_1", in2 := 15.0)
      { S7_Templates := "SrcType := Real" } LE_Contact(in1 := "m3_Obj_1", in2 := 15.2)
      Move(in := 1, out1 => "Tag_20")
   END_RUNG
   RUNG wire#powerrail
      { S7_Templates := "SrcType := Int" } EQ_Contact(in1 := "Tag_20", in2 := 0)
      wire#w1
      S_Coil( "10kg" )
   END_RUNG
   RUNG wire#w1
      R_Coil( "15Kg(1)" )
   END_RUNG
   RUNG wire#powerrail
      { S7_Templates := "SrcType := Int" } EQ_Contact(in1 := "Tag_20", in2 := 1)
      wire#w2
      S_Coil( "15Kg(1)" )
   END_RUNG
   RUNG wire#w2
      R_Coil( "10kg" )
   END_RUNG
   // the same network as SCL:
   IF ("m3_Obj_1" >= 10.0) AND ("m3_Obj_1" <= 10.2) THEN "Tag_20" := 0; END_IF;
   IF ("m3_Obj_1" >= 15.0) AND ("m3_Obj_1" <= 15.2) THEN "Tag_20" := 1; END_IF;
   IF "Tag_20" = 0 THEN
       "10kg" := TRUE;
       "15Kg(1)" := FALSE;
   END_IF;
   IF "Tag_20" = 1 THEN
       "15Kg(1)" := TRUE;
       "10kg" := FALSE;
   END_IF;
END_REGION

REGION Network 3
   #_w1 := "Start_Chiet" AND "Cb1";
   "FILLL"(EN := #_w1 AND "10kg",
           Level := 2.0,
           "1: Fill - 0: Dis" := 0,
           "Weight Obj" := "m3_Obj_1",
           Fill => "Discharge 3",
           ENO => #_w2);
   "T2".TON(IN := #_w2, PT := T#5S);
   "Continue with 10kg" := "T2".Q;
   "FILLL"(EN := #_w1 AND "15Kg(1)",
           Level := 2.0,
           "1: Fill - 0: Dis" := 0,
           "Weight Obj" := "m3_Obj_1",
           Fill => "Discharge 3",
           ENO => #_w3);
   "T3".TON(IN := #_w3, PT := T#7s);
   "Continue with 15kg" := "T3".Q;
   IF #_w1 AND ("Continue with 10kg" OR "Continue with 15kg") THEN "Discharge 3" := 0.0; END_IF;
END_REGION

REGION Network 4
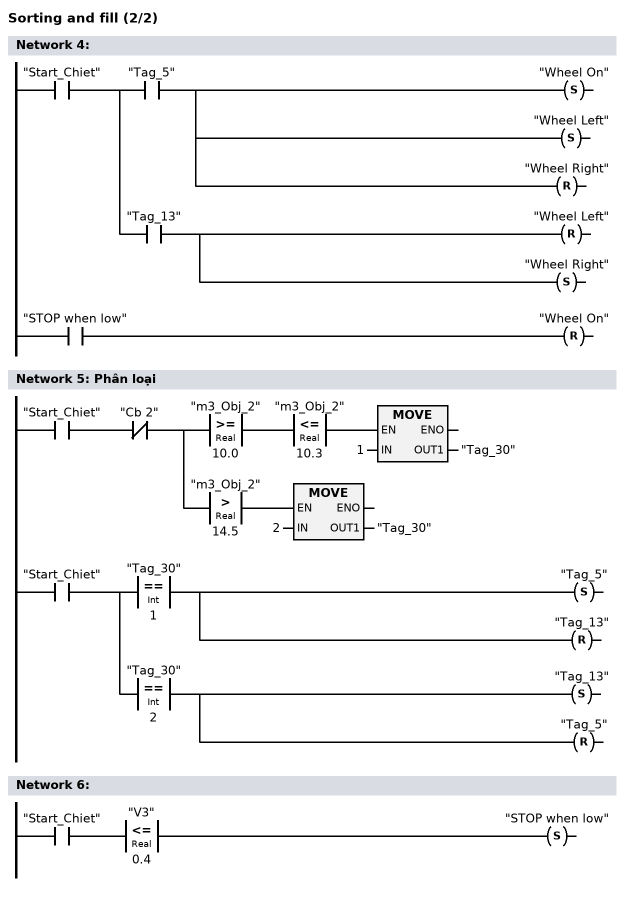
   RUNG wire#powerrail
      Contact( "Start_Chiet" )
      wire#w1
      Contact( "Tag_5" )
      wire#w2
      S_Coil( "Wheel On" )
   END_RUNG
   RUNG wire#w2
      S_Coil( "Wheel Left" )
   END_RUNG
   RUNG wire#w2
      R_Coil( "Wheel Right" )
   END_RUNG
   RUNG wire#w1
      Contact( "Tag_13" )
      wire#w3
      R_Coil( "Wheel Left" )
   END_RUNG
   RUNG wire#w3
      S_Coil( "Wheel Right" )
   END_RUNG
   RUNG wire#powerrail
      Contact( "STOP when low" )
      R_Coil( "Wheel On" )
   END_RUNG
   // the same network as SCL:
   IF "Start_Chiet" AND "Tag_5" THEN
       "Wheel On" := TRUE;
       "Wheel Left" := TRUE;
       "Wheel Right" := FALSE;
   END_IF;
   IF "Start_Chiet" AND "Tag_13" THEN
       "Wheel Left" := FALSE;
       "Wheel Right" := TRUE;
   END_IF;
   IF "STOP when low" THEN "Wheel On" := FALSE; END_IF;
END_REGION

REGION Network 5: Phân loại
   RUNG wire#powerrail
      Contact( "Start_Chiet" )
      I_Contact( "Cb 2" )
      wire#w1
      { S7_Templates := "SrcType := Real" } GE_Contact(in1 := "m3_Obj_2", in2 := 10.0)
      { S7_Templates := "SrcType := Real" } LE_Contact(in1 := "m3_Obj_2", in2 := 10.3)
      Move(in := 1, out1 => "Tag_30")
   END_RUNG
   RUNG wire#w1
      { S7_Templates := "SrcType := Real" } GT_Contact(in1 := "m3_Obj_2", in2 := 14.5)
      Move(in := 2, out1 => "Tag_30")
   END_RUNG
   RUNG wire#powerrail
      Contact( "Start_Chiet" )
      wire#w2
      { S7_Templates := "SrcType := Int" } EQ_Contact(in1 := "Tag_30", in2 := 1)
      wire#w3
      S_Coil( "Tag_5" )
   END_RUNG
   RUNG wire#w3
      R_Coil( "Tag_13" )
   END_RUNG
   RUNG wire#w2
      { S7_Templates := "SrcType := Int" } EQ_Contact(in1 := "Tag_30", in2 := 2)
      wire#w4
      S_Coil( "Tag_13" )
   END_RUNG
   RUNG wire#w4
      R_Coil( "Tag_5" )
   END_RUNG
   // the same network as SCL:
   #_w1 := "Start_Chiet" AND NOT "Cb 2";
   IF #_w1 AND ("m3_Obj_2" >= 10.0) AND ("m3_Obj_2" <= 10.3) THEN "Tag_30" := 1; END_IF;
   IF #_w1 AND ("m3_Obj_2" > 14.5) THEN "Tag_30" := 2; END_IF;
   IF "Start_Chiet" AND ("Tag_30" = 1) THEN
       "Tag_5" := TRUE;
       "Tag_13" := FALSE;
   END_IF;
   IF "Start_Chiet" AND ("Tag_30" = 2) THEN
       "Tag_13" := TRUE;
       "Tag_5" := FALSE;
   END_IF;
END_REGION

REGION Network 6
   RUNG wire#powerrail
      Contact( "Start_Chiet" )
      { S7_Templates := "SrcType := Real" } LE_Contact(in1 := "V3", in2 := 0.4)
      S_Coil( "STOP when low" )
   END_RUNG
   // the same network as SCL:
   IF "Start_Chiet" AND ("V3" <= 0.4) THEN "STOP when low" := TRUE; END_IF;
END_REGION
END_FUNCTION

FUNCTION "FILLL" : Void   // FC5, LAD
{ S7_Optimized_Access := 'TRUE' }
VERSION : 0.1
   VAR_INPUT
      Level : Real;
      "1: Fill - 0: Dis" : Bool;
      "Weight Obj" : Real;
   END_VAR
   VAR_OUTPUT
      Fill : Real;
   END_VAR
   VAR_TEMP
      "TG Voltage" : Real;
   END_VAR
BEGIN

REGION Network 1
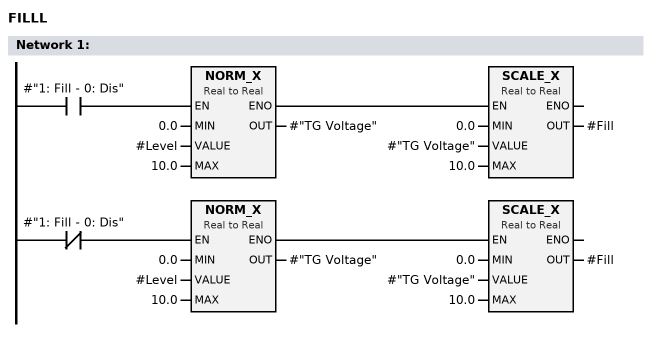
   RUNG wire#powerrail
      Contact( #"1: Fill - 0: Dis" )
      { S7_Templates := "[SrcType := Real, DestType := Real]" } Normalize(min := 0.0, value := #Level, max := 10.0, out => #"TG Voltage")
      { S7_Templates := "[SrcType := Real, DestType := Real]" } Scale(min := 0.0, value := #"TG Voltage", max := 10.0, out => #Fill)
   END_RUNG
   RUNG wire#powerrail
      I_Contact( #"1: Fill - 0: Dis" )
      { S7_Templates := "[SrcType := Real, DestType := Real]" } Normalize(min := 0.0, value := #Level, max := 10.0, out => #"TG Voltage")
      { S7_Templates := "[SrcType := Real, DestType := Real]" } Scale(min := 0.0, value := #"TG Voltage", max := 10.0, out => #Fill)
   END_RUNG
   // the same network as SCL:
   IF #"1: Fill - 0: Dis" THEN
       #"TG Voltage" := NORM_X(MIN := 0.0, VALUE := #Level, MAX := 10.0);
       #Fill := SCALE_X(MIN := 0.0, VALUE := #"TG Voltage", MAX := 10.0);
   END_IF;
   IF NOT #"1: Fill - 0: Dis" THEN
       #"TG Voltage" := NORM_X(MIN := 0.0, VALUE := #Level, MAX := 10.0);
       #Fill := SCALE_X(MIN := 0.0, VALUE := #"TG Voltage", MAX := 10.0);
   END_IF;
END_REGION
END_FUNCTION

FUNCTION "MHJ-PLC-Lab-Function-S71200" : Void   // FC9000, SCL
{ S7_Optimized_Access := 'TRUE' }
VERSION : 0.1
   VAR_TEMP
      rdTimeReturn : Int;
      outputTime : DTL;
      SyncVal : Byte;
      forVal : Int;
      forVal_2 : Int;
      Value : Byte;
   END_VAR
   VAR CONSTANT
      CompVal : Byte := 16#34;
      Value_01 : Byte := 16#11;
      Value_01_DW : DWord := 16#A165_D992;
      Value_02_DW : DWord := 16#58BE_4401;
   END_VAR
BEGIN

   #Value:=PEEK(area := 16#82,
        dbNumber := 0,
        byteOffset := 511);
   #Value := #Value + 1;

   POKE(area := 16#82,
        dbNumber := 0,
        byteOffset := 511,
        value := #Value);

   POKE(area:=16#81,
        dbNumber:=0,
        byteOffset:=1016,
        value:=#Value_01_DW);
   POKE(area := 16#81,
        dbNumber := 0,
        byteOffset := 1020,
        value := #Value_02_DW);

   POKE(area := 16#81,
        dbNumber := 0,
        byteOffset := 511,
        value := B#16#00);

   FOR #forVal := 0 TO 120 DO
       FOR #forVal_2:=0 TO 10 DO
           #rdTimeReturn:=RD_SYS_T(#outputTime);
           #rdTimeReturn := WR_SYS_T(#outputTime);
           #rdTimeReturn := RD_SYS_T(#outputTime);
           #rdTimeReturn := WR_SYS_T(#outputTime);
       END_FOR;
       #SyncVal:= PEEK(area := 16#81,
                      dbNumber := 0,
                      byteOffset := 511);
       IF #SyncVal = #CompVal THEN
          GOTO M_1;
       END_IF;
   END_FOR;
   RETURN;

   M_1:
   POKE(area := 16#81,
        dbNumber := 0,
        byteOffset := 511,
        value := B#16#0);
END_FUNCTION

ORGANIZATION_BLOCK "Main"   // OB1, LAD, ProgramCycle
TITLE = "Main Program Sweep (Cycle)"
{ S7_Optimized_Access := 'TRUE' }
VERSION : 0.1
   VAR_INPUT
      Initial_Call : Bool;   // Initial call of this OB
      Remanence : Bool;   // =True, if remanent data are available
   END_VAR
BEGIN

REGION Network 1: Konnektierungsbaustein für PLC-Lab
   // Im Netzwerk 1 wird der Konnektierungsbaustein für PLC-Lab aufgerufen.
   // Dieser Aufruf darf nicht entfernt werden!
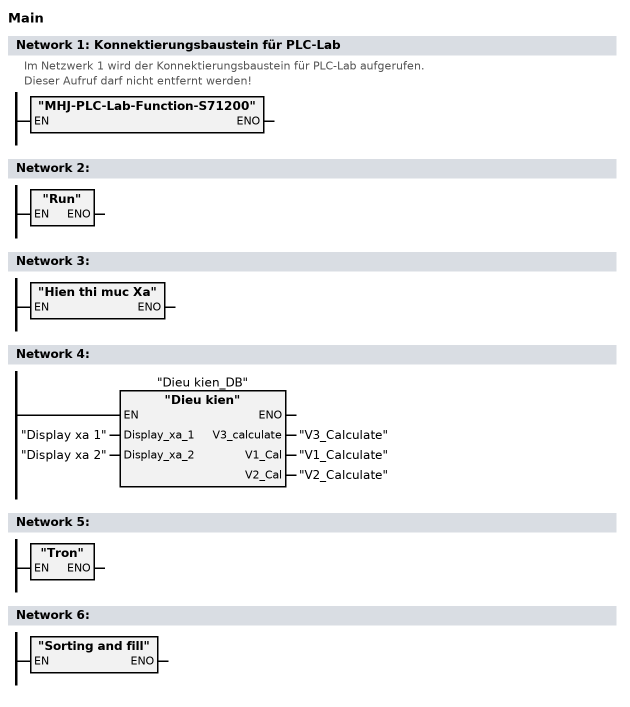
   RUNG wire#powerrail
      "MHJ-PLC-Lab-Function-S71200"()
   END_RUNG
   // the same network as SCL:
   "MHJ-PLC-Lab-Function-S71200"();
END_REGION

REGION Network 2
   RUNG wire#powerrail
      "Run"()
   END_RUNG
   // the same network as SCL:
   "Run"();
END_REGION

REGION Network 3
   RUNG wire#powerrail
      "Hien thi muc Xa"()
   END_RUNG
   // the same network as SCL:
   "Hien thi muc Xa"();
END_REGION

REGION Network 4
   RUNG wire#powerrail
      "Dieu kien_DB"(Display_xa_1 := "Display xa 1", Display_xa_2 := "Display xa 2", V3_calculate => "V3_Calculate", V1_Cal => "V1_Calculate", V2_Cal => "V2_Calculate")
   END_RUNG
   // the same network as SCL:
   "Dieu kien_DB"(Display_xa_1 := "Display xa 1",   // "Dieu kien"
                  Display_xa_2 := "Display xa 2",
                  V3_calculate => "V3_Calculate",
                  V1_Cal => "V1_Calculate",
                  V2_Cal => "V2_Calculate");
END_REGION

REGION Network 5
   RUNG wire#powerrail
      "Tron"()
   END_RUNG
   // the same network as SCL:
   "Tron"();
END_REGION

REGION Network 6
   RUNG wire#powerrail
      "Sorting and fill"()
   END_RUNG
   // the same network as SCL:
   "Sorting and fill"();
END_REGION
END_ORGANIZATION_BLOCK